FUNCTION_BLOCK XtsTrack EXTENDS CyclicBase IMPLEMENTS I_XtsTrack
VAR
	_MyInterface : I_TcIoXtsXpuTrack;
	XtsIoEnvInitialiseState : INT;
	MyPartCount : UDINT;
	Parts : REFERENCE TO ARRAY[1..TcIoXtsEnvironmentParameterList.MaxPartsPerTrack] OF ST_PartInfoItems;
	i : INT;
	_TrackLength: LREAL;
	_TrackIsClosed: BOOL;
	_OTCID : OTCID;
END_VAR

METHOD PUBLIC  Cycle : HRESULT
VAR_INPUT
END_VAR
Cycle := 2;
END_METHOD

METHOD Initialise : HRESULT
VAR_INPUT
END_VAR
CASE XtsIoEnvInitialiseState OF
	0:
		IF _MyInterface <> 0 THEN
			XtsIoEnvInitialiseState := 1;
		ELSE
			XtsIoEnvInitialiseState := 999;
		END_IF
	1:
		MyPartCount := _MyInterface.GetPartCount();
		XtsIoEnvInitialiseState := 2;
	2:
		XtsIoEnvInitialiseState := 3;
		Parts REF= _MyInterface.GetPartInfoItems();
		
	3:
		IF _MyInterface.P_IsInitialized THEN
			_TrackLength := _MyInterface.GetLength();
			_TrackIsClosed := _MyInterface.GetIsClosed();
			XtsIoEnvInitialiseState := 4;
		END_IF
	4:
		Initialise := 2;

END_CASE
END_METHOD

PROPERTY MyOTCID : OTCID
GET
MyOTCID := _OTCID;
END_GET
SET
_OTCID := MyOTCID;
END_SET
END_PROPERTY

PROPERTY MyXtsIoEnvInterface : I_TcIoXtsXpuTrack
GET
MyXtsIoEnvInterface := _MyInterface;
END_GET
SET
_MyInterface := MyXtsIoEnvInterface;
END_SET
END_PROPERTY

METHOD RemoveFromDetection : BOOL
VAR_INPUT
END_VAR
RemoveFromDetection := _MyInterface.SetIsIncludedInDetection(False);
END_METHOD

METHOD SetForDetection : BOOL
VAR_INPUT
END_VAR
SetForDetection := _MyInterface.SetIsIncludedInDetection(TRUE);
END_METHOD

PROPERTY TrackLength : MC_Lreal
GET
TrackLength := _MyInterface.GetLength();
END_GET
END_PROPERTY

END_FUNCTION_BLOCK

(* stored: Version 1.1.0.1
   POU XtsTrack: Id {0ed646c8-24dd-40d8-b451-d6e6a88b90d3}, SpecialFunc None
   Method Cycle: Id {753f4845-bb32-46bd-9afe-0c535a6bb9c5}
   Method Initialise: Id {b15a1974-ae41-45a0-b8ce-e38654aa0808}
   Property MyOTCID: Id {d34cfe46-c497-4e94-b74d-f99a6000b358}
   Get Get: Id {855c0947-7cfe-4f24-8259-2331fd728b0d}
   Set Set: Id {52d396c9-aa72-4a6c-b0f5-3d8704d35aca}
   Property MyXtsIoEnvInterface: Id {de406d6a-fb33-4758-a1bb-071b44e09534}
   Get Get: Id {29c07896-dd74-4eb2-b4f6-620c540248e5}
   Set Set: Id {efa5de65-cd69-47bf-b917-2b3471279c8e}
   Method RemoveFromDetection: Id {19fc9c17-6e83-4583-8661-ca0f3d7fbe00}
   Method SetForDetection: Id {2a4c4b2d-af72-4d4f-81aa-5409f825db3c}
   Property TrackLength: Id {f63b8800-afc4-4a64-a819-7bbd5ce82fd4}
   Get Get: Id {8c76ee9b-64b1-4933-b3fe-20fbe5dcfddc} *)
